{attribute 'qualified_only'}
VAR_GLOBAL
END_VAR

(* stored: Version 1.1.0.1, ProductVersion 3.1.4024.10
   GVL Parameter: Id {fb5b49eb-57ca-431c-a9c0-5270afaceaec} *)
